// Mitsubishi GX Works2 project: temp_hum   PLC: Q02/Q02H

PROGRAM TEMPHUM
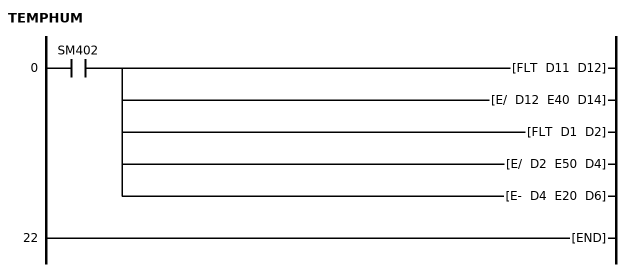
0     LD      SM402
      FLT     D11 D12
      E/      D12 E40 D14
      FLT     D1 D2
      E/      D2 E50 D4
      E-      D4 E20 D6
22    END
END_PROGRAM
